FUNCTION_BLOCK EL1712
VAR
	_io : EL1xx2_Data;
	{attribute addProperty Name "WcState"}
	_wcState : WcStateInputToggle;
	{attribute addProperty Name "Info data"}
	_infoData : InfoDataBase;
END_VAR

PROPERTY IO : REFERENCE TO EL1xx2_Data
GET
IO REF= _io;
END_GET
END_PROPERTY

PROPERTY WcState : REFERENCE TO WcStateInputToggle
GET
WcState REF= _wcState;
END_GET
END_PROPERTY

END_FUNCTION_BLOCK

(* stored: Version 1.1.0.1, ProductVersion 3.1.4024.9
   POU EL1712: Id {d183578d-1087-06fc-2514-62d750b466e3}, SpecialFunc None
   Property IO: Id {6992dab4-1025-05a7-2e62-8f2c2dda7fe6}
   Get Get: Id {f018fc07-fa6b-096d-1a14-767eac5656c6}
   Property WcState: Id {a178a64f-7db2-07b6-060f-e91fd42ce609}
   Get Get: Id {c1469bb4-98ac-048f-2ca0-c5155bbc6def} *)
